// TIA Portal V16 export
// export: Created 2020-03-22T19:23:53.3719267Z, ExportSetting WithDefaults, DisplayName Totally Integrated Automation Portal, DisplayVersion V16, DisplayName TIA Portal Version Control Interface, DisplayVersion V16, DisplayName TIA Portal Openness, DisplayVersion V16, DisplayName TIA Portal Teamcenter Gateway, DisplayVersion V16, DisplayName SINAMICS Startdrive Advanced, DisplayVersion V16 Update 1, DisplayName SINAMICS Startdrive G130, G150, S120, S150, SINAMICS MV, S210, DisplayVersion V16 Update 1, DisplayName SINAMICS Startdrive G110M, G120, G120C, G120D, G120P, DisplayVersion V16 Update 1, DisplayName STEP 7 Professional, DisplayVersion V16, DisplayName STEP 7 Safety, DisplayVersion V16, DisplayName WinCC Professional, DisplayVersion V16
FUNCTION_BLOCK "TX-AI"   // FB804, LAD
{ S7_Optimized_Access := 'TRUE' }
VERSION : 1.0
// stored: AutoNumber false, IsIECCheckEnabled false, IsRetainMemResEnabled false, MemoryReserve 100, SetENOAutomatically false, UDAEnableTagReadback false
   VAR_INPUT
      Mode { ExternalAccessible := 'False'; ExternalVisible := 'False'; ExternalWritable := 'False'} : Int;   // TX Mode - 0 = 4-20 mA / 1 = Int Math (RTD/TC) / 3 = SQRT / 6 = Vortex
      RAIVI { ExternalAccessible := 'False'; ExternalVisible := 'False'; ExternalWritable := 'False'} : Int;   // Raw Analog Input Value INT
      RAIVR { ExternalAccessible := 'False'; ExternalVisible := 'False'; ExternalWritable := 'False'} : Real;   // Raw Analog Input Value REAL
   END_VAR
   VAR_OUTPUT
      SAI : Real;   // Compensated Scaled Analog Value
   END_VAR
   VAR
      HMI : Struct   // Alarms
         Status : Struct
            USAV : Real;   // Uncompensated Scaled Analog Value
            TCV : Real;   // Temperature Compensation Value
            PCV : Real;   // Pressure Compensation Value
            NV : Real;   // Normalized Value
         END_STRUCT;
         Alarm : Struct   // Alarms
            AHHH : Bool;   // Alarm - High High High
            AHH : Bool;   // Alarm - High High
            AH : Bool;   // Alarm - High
            AL : Bool;   // Alarm - Low
            ALL : Bool;   // Alarm - Low Low
            ALLL : Bool;   // Alarm - Low Low Low
            "OR" : Bool;   // Alarm Over Range
            UR : Bool;   // Alarm Under Range
            Fault : Bool;   // Alarm Fault
            SUB : Bool;   // Fault detected and output value is the defined subsitution value
            CH_Fault : Bool;
         END_STRUCT;
         Config : Struct   // Settings
            RIMXV : Real := 27648.0;   // Raw Input Maximum Value (Used for Sqrt)
            RIMNV : Real;   // Raw Input Minimum Value (Used for Sqrt)
            ESMXV : Real := 100.0;   // Engineering/Scaled Maximum Value
            ESMNV : Real;   // Engineering/Scaled Minimum Value
            COV : Bool;   // Clamp Output Value
            OV : Real;   // Offset Value
            SAM : Bool;   // Substitution Activation Mode
            SAV : Real := -999999.0;   // Substitution Value during a limit input value trip
            CE : Struct   // Compensation Equation
               TC : Real := 460.0;   // Temperature Constant
               PC : Real := 14.7;   // Pressure Constant
               TR : Real := 1.0;   // Temperature Reference
               TA : Real := 1.0;   // Temperature Actual
               PR : Real := 1.0;   // Pressure Reference
               PA : Real := 1.0;   // Pressure Actual
            END_STRUCT;
            SP : Struct   // Setpoints
               Limits : Struct
                  HHH : Real := 95.0;   // HHH Limit Setpoint
                  HH : Real := 90.0;   // HH Limit Setpoint
                  H : Real := 80.0;   // HH Limit Setpoint
                  L : Real := 20.0;   // L Limit Setpoint
                  LL : Real := 10.0;   // LL Limit Setpoint
                  LLL : Real := 5.0;   // LLL Limit Setpoint
                  "OR" : Real := 5.0;   // Over range value
                  UR : Real := 5.0;   // Under range value
               END_STRUCT;
               HYS : Struct   // Hysteresis
                  Global : Real;   // Hysteresis global value, only valid when greater than or equal to 0
                  HHH : Real := 1.0;   // Hysteresis Setpoint - High High High
                  HH : Real := 1.0;   // Hysteresis Setpoint - High High
                  H : Real := 1.0;   // Hysteresis Setpoint - High
                  L : Real := 1.0;   // Hysteresis Setpoint - Low
                  LL : Real := 1.0;   // Hysteresis Setpoint - Low Low
                  LLL : Real := 1.0;   // Hysteresis Setpoint - Low Low Low
                  "OR" : Real := 1.0;   // Hysteresis Setpoint - Over Range
                  UR : Real := 1.0;   // Hysteresis Setpoint - Under Range
               END_STRUCT;
               SUB_ON : Bool;   // Substitution Activation
            END_STRUCT;
            PT : Struct   // Setpoints
               HLD : Struct   // Hold
                  Global : Time;   // Hold PT global value, only valid when not equal to 0
                  AHHH : Time := T#1S;   // Alarm Debounce
                  AHH : Time := T#1S;   // Alarm Debounce
                  AH : Time := T#1S;   // Alarm Debounce
                  AL : Time := T#1S;   // Alarm Debounce
                  ALL : Time := T#1S;   // Alarm Debounce
                  ALLL : Time := T#1S;   // Alarm Debounce
                  "OR" : Time := T#1S;   // Over range hold
                  UR : Time := T#1S;   // Under range hold
               END_STRUCT;
               DBNC : Struct   // Debounce
                  Global : Time;   // Debounce PT global value, only valid when not equal to 0
                  AHHH : Time := T#1S;   // Alarm Debounce
                  AHH : Time := T#1S;   // Alarm Debounce
                  AH : Time := T#1S;   // Alarm Debounce
                  AL : Time := T#1S;   // Alarm Debounce
                  ALL : Time := T#1S;   // Alarm Debounce
                  ALLL : Time := T#1S;   // Alarm Debounce
                  "OR" : Time := T#1S;   // Over range debounce
                  UR : Time := T#1S;   // Under range debounce
               END_STRUCT;
            END_STRUCT;
         END_STRUCT;
         Diag : Struct   // Diagnostics
            SV : Real;   // Simulation Value
         END_STRUCT;
      END_STRUCT;
      Admin : Struct   // Admin configurations
         SCL : Struct   // Scale Values
            RDP : Real := 10.0;   // RTD Decimal Places
            RRIMD : Real := 1.0;   // Raw Real input Math divider
            "OR" : Real;   // Over Range Value
            UR : Real;   // Under Range Value
            SAIV : Real;   // Scaled Analog Input Value
         END_STRUCT;
         HYS : Struct   // Hysteresis - Computed Values
            "OR" : Real;   // Hysteresis Value - Over Range
            UR : Real;   // Hysteresis Value - Under Range
         END_STRUCT;
      END_STRUCT;
      OR_DB { ExternalAccessible := 'False'; ExternalVisible := 'False'; ExternalWritable := 'False'} : TON_TIME;   // Over Range Debounce
      UR_DB { ExternalAccessible := 'False'; ExternalVisible := 'False'; ExternalWritable := 'False'} : TON_TIME;   // Under Range DB
      OR_HLD { ExternalAccessible := 'False'; ExternalVisible := 'False'; ExternalWritable := 'False'} : TOF_TIME;   // Over Range Hold
      UR_HLD { ExternalAccessible := 'False'; ExternalVisible := 'False'; ExternalWritable := 'False'} : TOF_TIME;   // Under Range Hold
      HHHA { ExternalAccessible := 'False'; ExternalVisible := 'False'; ExternalWritable := 'False'} : "HLR";   // High High High Alarm
      HHA { ExternalAccessible := 'False'; ExternalVisible := 'False'; ExternalWritable := 'False'} : "HLR";   // High High Alarm
      HA { ExternalAccessible := 'False'; ExternalVisible := 'False'; ExternalWritable := 'False'} : "HLR";   // High Alarm
      LA { ExternalAccessible := 'False'; ExternalVisible := 'False'; ExternalWritable := 'False'} : "LLR";   // Low Alarm
      LLA { ExternalAccessible := 'False'; ExternalVisible := 'False'; ExternalWritable := 'False'} : "LLR";   // Low Low Alarm
      LLLA { ExternalAccessible := 'False'; ExternalVisible := 'False'; ExternalWritable := 'False'} : "LLR";   // Low Low Low Alarm
      molActual { ExternalAccessible := 'False'; ExternalVisible := 'False'; ExternalWritable := 'False'} : Real := 1.0;
      molDesign { ExternalAccessible := 'False'; ExternalVisible := 'False'; ExternalWritable := 'False'} : Real := 1.0;
   END_VAR
   VAR_TEMP
      RAIDI : DInt;   // Raw Analog Input DINT
      RAIR : Real;   // Raw Analog Input REAL
      RAIAV : Real;   // Raw Analog Input Absolute Value
      RAISRV : Real;   // Raw Analog Input Square Root Value
      RAIVS : Real;   // Raw Analog Input Value Scaler
      TCRE : Real;   // Temperature Compensation Reference Equation
      TCAE : Real;   // Temperature Compensation Actual Equation
      PCRE : Real;   // Pressure Compensation Reference Equation
      PCAE : Real;   // Pressure Compensation Actual Equation
      TPCV : Real;   // Temperature Pressure Compensation Value
      MWCV : Real;   // Mol Weight Compensation Value
      TPMCV : Real;   // Temperature Pressure Mol Compensation Value
      sqrtSaiv : Real;   // SCALED ANALOG INT VALUE TO BE SQRT'D
      rawValue : Int;
      dummy : Bool;
      sqrt01 : Real;
      RAIVR_1 : DInt;
      RAIVR_1_1 : Real;
   END_VAR
   VAR_TEMP   // added for the SCL form of the ladder/FBD networks
      _w1 : Bool;
      _w2 : Bool;
   END_VAR
BEGIN

REGION Network 1: Transmitter Mode 1 = Int Math or RTD
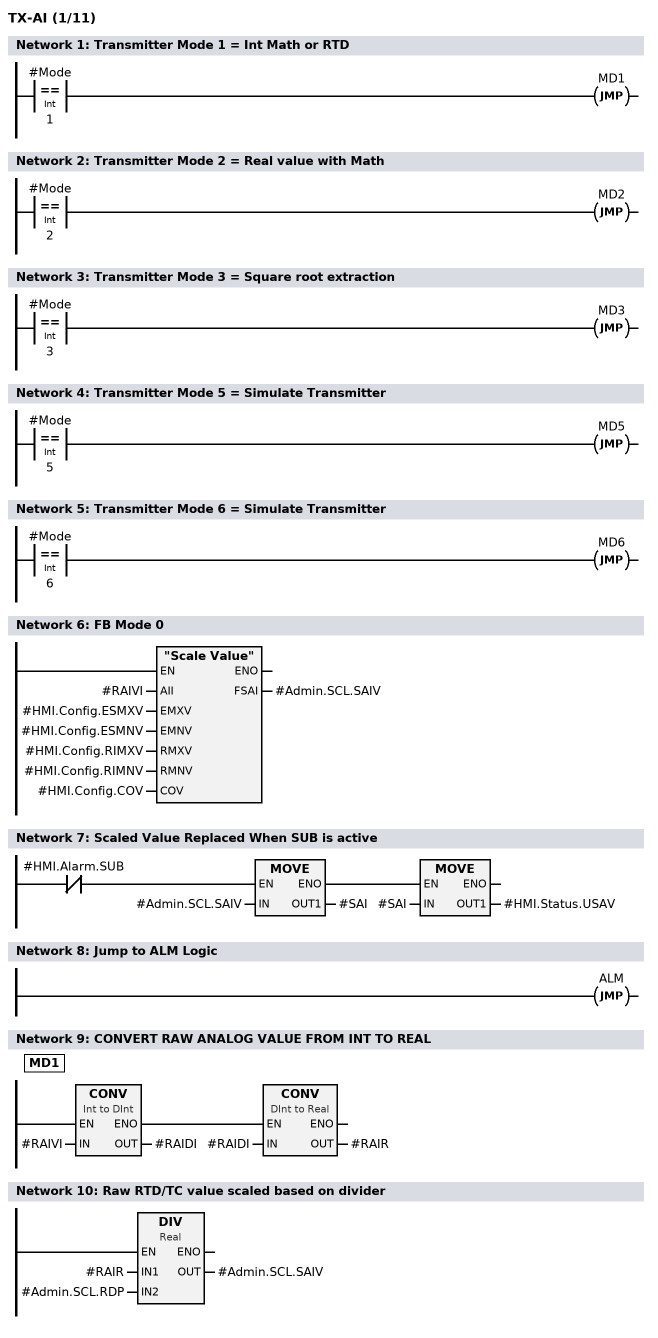
   RUNG wire#powerrail
      { S7_Templates := "SrcType := Int" } EQ_Contact(in1 := #Mode, in2 := 1)
      JumpCoil( MD1 )
   END_RUNG
   // the same network as SCL:
   IF #Mode = 1 THEN GOTO MD1; END_IF;
END_REGION

REGION Network 2: Transmitter Mode 2 = Real value with Math
   RUNG wire#powerrail
      { S7_Templates := "SrcType := Int" } EQ_Contact(in1 := #Mode, in2 := 2)
      JumpCoil( MD2 )
   END_RUNG
   // the same network as SCL:
   IF #Mode = 2 THEN GOTO MD2; END_IF;
END_REGION

REGION Network 3: Transmitter Mode 3 = Square root extraction
   RUNG wire#powerrail
      { S7_Templates := "SrcType := Int" } EQ_Contact(in1 := #Mode, in2 := 3)
      JumpCoil( MD3 )
   END_RUNG
   // the same network as SCL:
   IF #Mode = 3 THEN GOTO MD3; END_IF;
END_REGION

REGION Network 4: Transmitter Mode 5 = Simulate Transmitter
   RUNG wire#powerrail
      { S7_Templates := "SrcType := Int" } EQ_Contact(in1 := #Mode, in2 := 5)
      JumpCoil( MD5 )
   END_RUNG
   // the same network as SCL:
   IF #Mode = 5 THEN GOTO MD5; END_IF;
END_REGION

REGION Network 5: Transmitter Mode 6 = Simulate Transmitter
   RUNG wire#powerrail
      { S7_Templates := "SrcType := Int" } EQ_Contact(in1 := #Mode, in2 := 6)
      JumpCoil( MD6 )
   END_RUNG
   // the same network as SCL:
   IF #Mode = 6 THEN GOTO MD6; END_IF;
END_REGION

REGION Network 6: FB Mode 0
   RUNG wire#powerrail
      "Scale Value"(AII := #RAIVI, EMXV := #HMI.Config.ESMXV, EMNV := #HMI.Config.ESMNV, RMXV := #HMI.Config.RIMXV, RMNV := #HMI.Config.RIMNV, COV := #HMI.Config.COV, FSAI => #Admin.SCL.SAIV)
   END_RUNG
   // the same network as SCL:
   "Scale Value"(AII := #RAIVI,
                 EMXV := #HMI.Config.ESMXV,
                 EMNV := #HMI.Config.ESMNV,
                 RMXV := #HMI.Config.RIMXV,
                 RMNV := #HMI.Config.RIMNV,
                 COV := #HMI.Config.COV,
                 FSAI => #Admin.SCL.SAIV);
END_REGION

REGION Network 7: Scaled Value Replaced When SUB is active
   RUNG wire#powerrail
      I_Contact( #HMI.Alarm.SUB )
      { S7_GenerateENO := "TRUE" } Move(in := #Admin.SCL.SAIV, out1 => #SAI)
      { S7_GenerateENO := "TRUE" } Move(in := #SAI, out1 => #HMI.Status.USAV)
   END_RUNG
   // the same network as SCL:
   // ENO of a box is taken as its EN; it also drops when the box reports an error
   IF NOT #HMI.Alarm.SUB THEN
       #SAI := #Admin.SCL.SAIV;
       #HMI.Status.USAV := #SAI;
   END_IF;
END_REGION

REGION Network 8: Jump to ALM Logic
   RUNG wire#powerrail
      JumpCoil( ALM )
   END_RUNG
   // the same network as SCL:
   GOTO ALM;
END_REGION

REGION Network 9: CONVERT RAW ANALOG VALUE FROM INT TO REAL
   Label( MD1 )
   RUNG wire#powerrail
      { S7_Templates := "[SrcType := Int, DestType := DInt]"; S7_GenerateENO := "TRUE" } Convert(in := #RAIVI, out => #RAIDI)
      { S7_Templates := "[SrcType := DInt, DestType := Real]"; S7_GenerateENO := "TRUE" } Convert(in := #RAIDI, out => #RAIR)
   END_RUNG
   // the same network as SCL:
   // ENO of a box is taken as its EN; it also drops when the box reports an error
   MD1:
   #RAIDI := INT_TO_DINT(#RAIVI);
   #RAIR := DINT_TO_REAL(#RAIDI);
END_REGION

REGION Network 10: Raw RTD/TC value scaled based on divider
   RUNG wire#powerrail
      { S7_Templates := "SrcType := Real"; S7_GenerateENO := "TRUE" } Div(in1 := #RAIR, in2 := #Admin.SCL.RDP, out => #Admin.SCL.SAIV)
   END_RUNG
   // the same network as SCL:
   #Admin.SCL.SAIV := #RAIR / #Admin.SCL.RDP;
END_REGION

REGION Network 11: Scaled Value Replaced When SUB is active
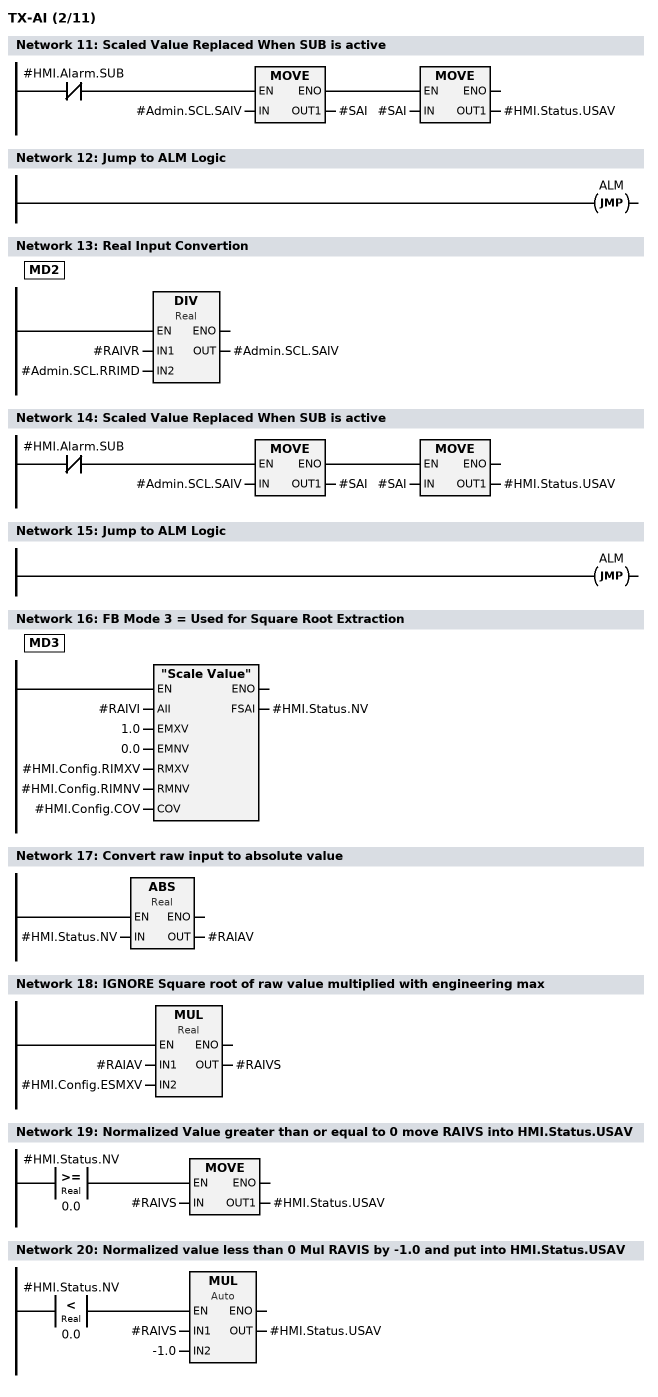
   RUNG wire#powerrail
      I_Contact( #HMI.Alarm.SUB )
      { S7_GenerateENO := "TRUE" } Move(in := #Admin.SCL.SAIV, out1 => #SAI)
      Move(in := #SAI, out1 => #HMI.Status.USAV)
   END_RUNG
   // the same network as SCL:
   // ENO of a box is taken as its EN; it also drops when the box reports an error
   IF NOT #HMI.Alarm.SUB THEN
       #SAI := #Admin.SCL.SAIV;
       #HMI.Status.USAV := #SAI;
   END_IF;
END_REGION

REGION Network 12: Jump to ALM Logic
   RUNG wire#powerrail
      JumpCoil( ALM )
   END_RUNG
   // the same network as SCL:
   GOTO ALM;
END_REGION

REGION Network 13: Real Input Convertion
   Label( MD2 )
   RUNG wire#powerrail
      { S7_Templates := "SrcType := Real"; S7_GenerateENO := "TRUE" } Div(in1 := #RAIVR, in2 := #Admin.SCL.RRIMD, out => #Admin.SCL.SAIV)
   END_RUNG
   // the same network as SCL:
   MD2:
   #Admin.SCL.SAIV := #RAIVR / #Admin.SCL.RRIMD;
END_REGION

REGION Network 14: Scaled Value Replaced When SUB is active
   RUNG wire#powerrail
      I_Contact( #HMI.Alarm.SUB )
      { S7_GenerateENO := "TRUE" } Move(in := #Admin.SCL.SAIV, out1 => #SAI)
      Move(in := #SAI, out1 => #HMI.Status.USAV)
   END_RUNG
   // the same network as SCL:
   // ENO of a box is taken as its EN; it also drops when the box reports an error
   IF NOT #HMI.Alarm.SUB THEN
       #SAI := #Admin.SCL.SAIV;
       #HMI.Status.USAV := #SAI;
   END_IF;
END_REGION

REGION Network 15: Jump to ALM Logic
   RUNG wire#powerrail
      JumpCoil( ALM )
   END_RUNG
   // the same network as SCL:
   GOTO ALM;
END_REGION

REGION Network 16: FB Mode 3 = Used for Square Root Extraction
   Label( MD3 )
   RUNG wire#powerrail
      "Scale Value"(AII := #RAIVI, EMXV := 1.0, EMNV := 0.0, RMXV := #HMI.Config.RIMXV, RMNV := #HMI.Config.RIMNV, COV := #HMI.Config.COV, FSAI => #HMI.Status.NV)
   END_RUNG
   // the same network as SCL:
   MD3:
   "Scale Value"(AII := #RAIVI,
                 EMXV := 1.0,
                 EMNV := 0.0,
                 RMXV := #HMI.Config.RIMXV,
                 RMNV := #HMI.Config.RIMNV,
                 COV := #HMI.Config.COV,
                 FSAI => #HMI.Status.NV);
END_REGION

REGION Network 17: Convert raw input to absolute value
   RUNG wire#powerrail
      { S7_Templates := "SrcType := Real"; S7_GenerateENO := "TRUE" } Abs(in := #HMI.Status.NV, out => #RAIAV)
   END_RUNG
   // the same network as SCL:
   #RAIAV := ABS(#HMI.Status.NV);
END_REGION

REGION Network 18: IGNORE Square root of raw value multiplied with engineering max
   RUNG wire#powerrail
      { S7_Templates := "SrcType := Real"; S7_GenerateENO := "TRUE" } Mul(in1 := #RAIAV, in2 := #HMI.Config.ESMXV, out => #RAIVS)
   END_RUNG
   // the same network as SCL:
   #RAIVS := #RAIAV * #HMI.Config.ESMXV;
END_REGION

REGION Network 19: Normalized Value greater than or equal to 0 move RAIVS into HMI.Status.USAV
   RUNG wire#powerrail
      { S7_Templates := "SrcType := Real" } GE_Contact(in1 := #HMI.Status.NV, in2 := 0.0)
      { S7_GenerateENO := "TRUE" } Move(in := #RAIVS, out1 => #HMI.Status.USAV)
   END_RUNG
   // the same network as SCL:
   IF #HMI.Status.NV >= 0.0 THEN #HMI.Status.USAV := #RAIVS; END_IF;
END_REGION

REGION Network 20: Normalized value less than 0 Mul RAVIS by -1.0 and put into HMI.Status.USAV
   RUNG wire#powerrail
      { S7_Templates := "SrcType := Real" } LT_Contact(in1 := #HMI.Status.NV, in2 := 0.0)
      { S7_GenerateENO := "TRUE" } Mul(in1 := #RAIVS, in2 := -1.0, out => #HMI.Status.USAV)
   END_RUNG
   // the same network as SCL:
   IF #HMI.Status.NV < 0.0 THEN #HMI.Status.USAV := #RAIVS * (-1.0); END_IF;
END_REGION

REGION Network 21: Temperature Compensation Equation Step 1
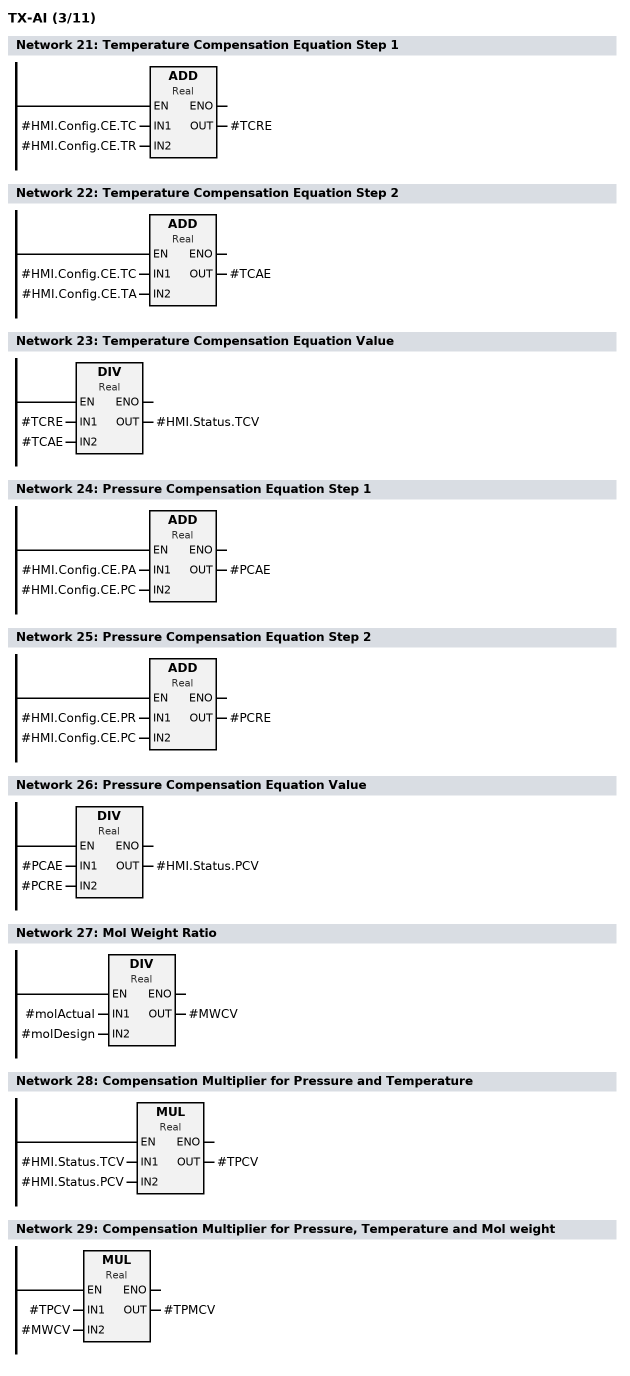
   RUNG wire#powerrail
      { S7_Templates := "SrcType := Real"; S7_GenerateENO := "TRUE" } Add(in1 := #HMI.Config.CE.TC, in2 := #HMI.Config.CE.TR, out => #TCRE)
   END_RUNG
   // the same network as SCL:
   #TCRE := #HMI.Config.CE.TC + #HMI.Config.CE.TR;
END_REGION

REGION Network 22: Temperature Compensation Equation Step 2
   RUNG wire#powerrail
      { S7_Templates := "SrcType := Real"; S7_GenerateENO := "TRUE" } Add(in1 := #HMI.Config.CE.TC, in2 := #HMI.Config.CE.TA, out => #TCAE)
   END_RUNG
   // the same network as SCL:
   #TCAE := #HMI.Config.CE.TC + #HMI.Config.CE.TA;
END_REGION

REGION Network 23: Temperature Compensation Equation Value
   RUNG wire#powerrail
      { S7_Templates := "SrcType := Real"; S7_GenerateENO := "TRUE" } Div(in1 := #TCRE, in2 := #TCAE, out => #HMI.Status.TCV)
   END_RUNG
   // the same network as SCL:
   #HMI.Status.TCV := #TCRE / #TCAE;
END_REGION

REGION Network 24: Pressure Compensation Equation Step 1
   RUNG wire#powerrail
      { S7_Templates := "SrcType := Real"; S7_GenerateENO := "TRUE" } Add(in1 := #HMI.Config.CE.PA, in2 := #HMI.Config.CE.PC, out => #PCAE)
   END_RUNG
   // the same network as SCL:
   #PCAE := #HMI.Config.CE.PA + #HMI.Config.CE.PC;
END_REGION

REGION Network 25: Pressure Compensation Equation Step 2
   RUNG wire#powerrail
      { S7_Templates := "SrcType := Real"; S7_GenerateENO := "TRUE" } Add(in1 := #HMI.Config.CE.PR, in2 := #HMI.Config.CE.PC, out => #PCRE)
   END_RUNG
   // the same network as SCL:
   #PCRE := #HMI.Config.CE.PR + #HMI.Config.CE.PC;
END_REGION

REGION Network 26: Pressure Compensation Equation Value
   RUNG wire#powerrail
      { S7_Templates := "SrcType := Real"; S7_GenerateENO := "TRUE" } Div(in1 := #PCAE, in2 := #PCRE, out => #HMI.Status.PCV)
   END_RUNG
   // the same network as SCL:
   #HMI.Status.PCV := #PCAE / #PCRE;
END_REGION

REGION Network 27: Mol Weight Ratio
   RUNG wire#powerrail
      { S7_Templates := "SrcType := Real"; S7_GenerateENO := "TRUE" } Div(in1 := #molActual, in2 := #molDesign, out => #MWCV)
   END_RUNG
   // the same network as SCL:
   #MWCV := #molActual / #molDesign;
END_REGION

REGION Network 28: Compensation Multiplier for Pressure and Temperature
   RUNG wire#powerrail
      { S7_Templates := "SrcType := Real"; S7_GenerateENO := "TRUE" } Mul(in1 := #HMI.Status.TCV, in2 := #HMI.Status.PCV, out => #TPCV)
   END_RUNG
   // the same network as SCL:
   #TPCV := #HMI.Status.TCV * #HMI.Status.PCV;
END_REGION

REGION Network 29: Compensation Multiplier for Pressure, Temperature and Mol weight
   RUNG wire#powerrail
      { S7_Templates := "SrcType := Real"; S7_GenerateENO := "TRUE" } Mul(in1 := #TPCV, in2 := #MWCV, out => #TPMCV)
   END_RUNG
   // the same network as SCL:
   #TPMCV := #TPCV * #MWCV;
END_REGION

REGION Network 30: Compensated Analog Value
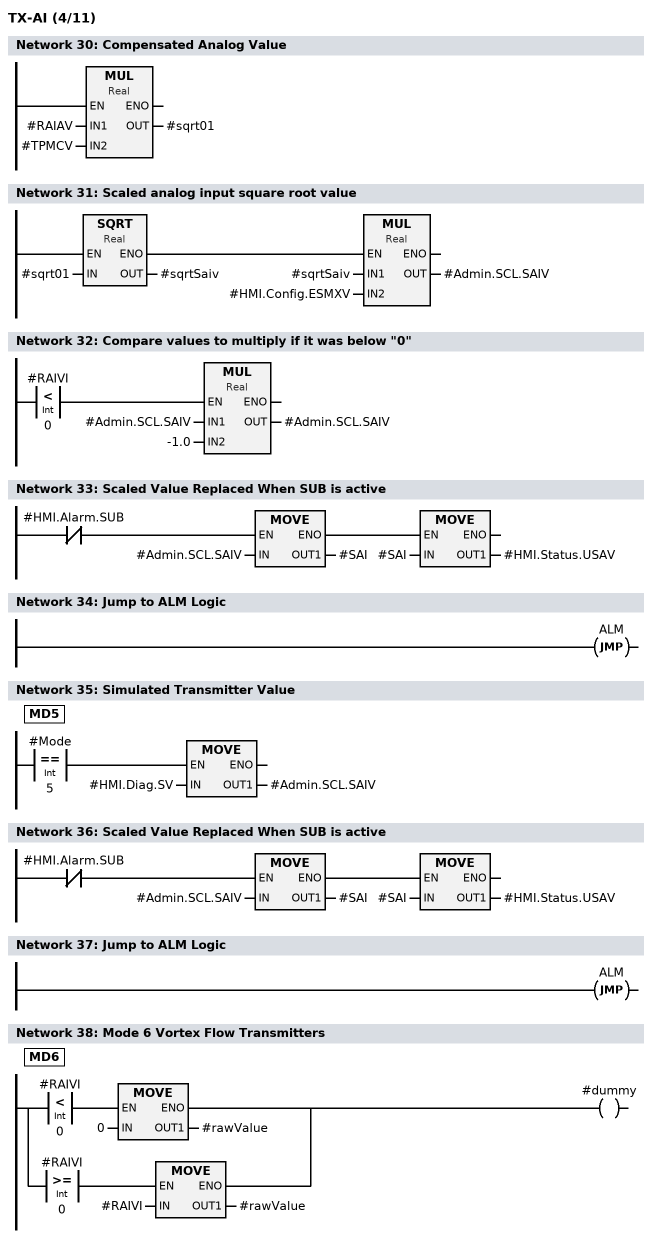
   RUNG wire#powerrail
      { S7_Templates := "SrcType := Real"; S7_GenerateENO := "TRUE" } Mul(in1 := #RAIAV, in2 := #TPMCV, out => #sqrt01)
   END_RUNG
   // the same network as SCL:
   #sqrt01 := #RAIAV * #TPMCV;
END_REGION

REGION Network 31: Scaled analog input square root value
   // ENO of a box is taken as its EN; it also drops when the box reports an error
   #sqrtSaiv := SQRT(#sqrt01);
   #Admin.SCL.SAIV := #sqrtSaiv * #HMI.Config.ESMXV;
END_REGION

REGION Network 32: Compare values to multiply if it was below "0"
   RUNG wire#powerrail
      { S7_Templates := "SrcType := Int" } LT_Contact(in1 := #RAIVI, in2 := 0)
      { S7_Templates := "SrcType := Real"; S7_GenerateENO := "TRUE" } Mul(in1 := #Admin.SCL.SAIV, in2 := -1.0, out => #Admin.SCL.SAIV)
   END_RUNG
   // the same network as SCL:
   IF #RAIVI < 0 THEN #Admin.SCL.SAIV := #Admin.SCL.SAIV * (-1.0); END_IF;
END_REGION

REGION Network 33: Scaled Value Replaced When SUB is active
   RUNG wire#powerrail
      I_Contact( #HMI.Alarm.SUB )
      { S7_GenerateENO := "TRUE" } Move(in := #Admin.SCL.SAIV, out1 => #SAI)
      { S7_GenerateENO := "TRUE" } Move(in := #SAI, out1 => #HMI.Status.USAV)
   END_RUNG
   // the same network as SCL:
   // ENO of a box is taken as its EN; it also drops when the box reports an error
   IF NOT #HMI.Alarm.SUB THEN
       #SAI := #Admin.SCL.SAIV;
       #HMI.Status.USAV := #SAI;
   END_IF;
END_REGION

REGION Network 34: Jump to ALM Logic
   RUNG wire#powerrail
      JumpCoil( ALM )
   END_RUNG
   // the same network as SCL:
   GOTO ALM;
END_REGION

REGION Network 35: Simulated Transmitter Value
   Label( MD5 )
   RUNG wire#powerrail
      { S7_Templates := "SrcType := Int" } EQ_Contact(in1 := #Mode, in2 := 5)
      { S7_GenerateENO := "TRUE" } Move(in := #HMI.Diag.SV, out1 => #Admin.SCL.SAIV)
   END_RUNG
   // the same network as SCL:
   MD5:
   IF #Mode = 5 THEN #Admin.SCL.SAIV := #HMI.Diag.SV; END_IF;
END_REGION

REGION Network 36: Scaled Value Replaced When SUB is active
   RUNG wire#powerrail
      I_Contact( #HMI.Alarm.SUB )
      { S7_GenerateENO := "TRUE" } Move(in := #Admin.SCL.SAIV, out1 => #SAI)
      { S7_GenerateENO := "TRUE" } Move(in := #SAI, out1 => #HMI.Status.USAV)
   END_RUNG
   // the same network as SCL:
   // ENO of a box is taken as its EN; it also drops when the box reports an error
   IF NOT #HMI.Alarm.SUB THEN
       #SAI := #Admin.SCL.SAIV;
       #HMI.Status.USAV := #SAI;
   END_IF;
END_REGION

REGION Network 37: Jump to ALM Logic
   RUNG wire#powerrail
      JumpCoil( ALM )
   END_RUNG
   // the same network as SCL:
   GOTO ALM;
END_REGION

REGION Network 38: Mode 6 Vortex Flow Transmitters
   Label( MD6 )
   RUNG wire#powerrail
      { S7_Templates := "SrcType := Int" } LT_Contact(in1 := #RAIVI, in2 := 0)
      { S7_GenerateENO := "TRUE" } Move(in := 0, out1 => #rawValue)
      wire#w1
      Coil( #dummy )
   END_RUNG
   RUNG wire#powerrail
      { S7_Templates := "SrcType := Int" } GE_Contact(in1 := #RAIVI, in2 := 0)
      { S7_GenerateENO := "TRUE" } Move(in := #RAIVI, out1 => #rawValue)
   END_RUNG wire#w1
   // the same network as SCL:
   // ENO of a box is taken as its EN; it also drops when the box reports an error
   MD6:
   #_w1 := #RAIVI < 0;
   IF #_w1 THEN #rawValue := 0; END_IF;
   #_w2 := #RAIVI >= 0;
   IF #_w2 THEN #rawValue := #RAIVI; END_IF;
   #dummy := #_w1 OR #_w2;
END_REGION

REGION Network 39: Normalize signal 4-20mA to 0-1 ratio
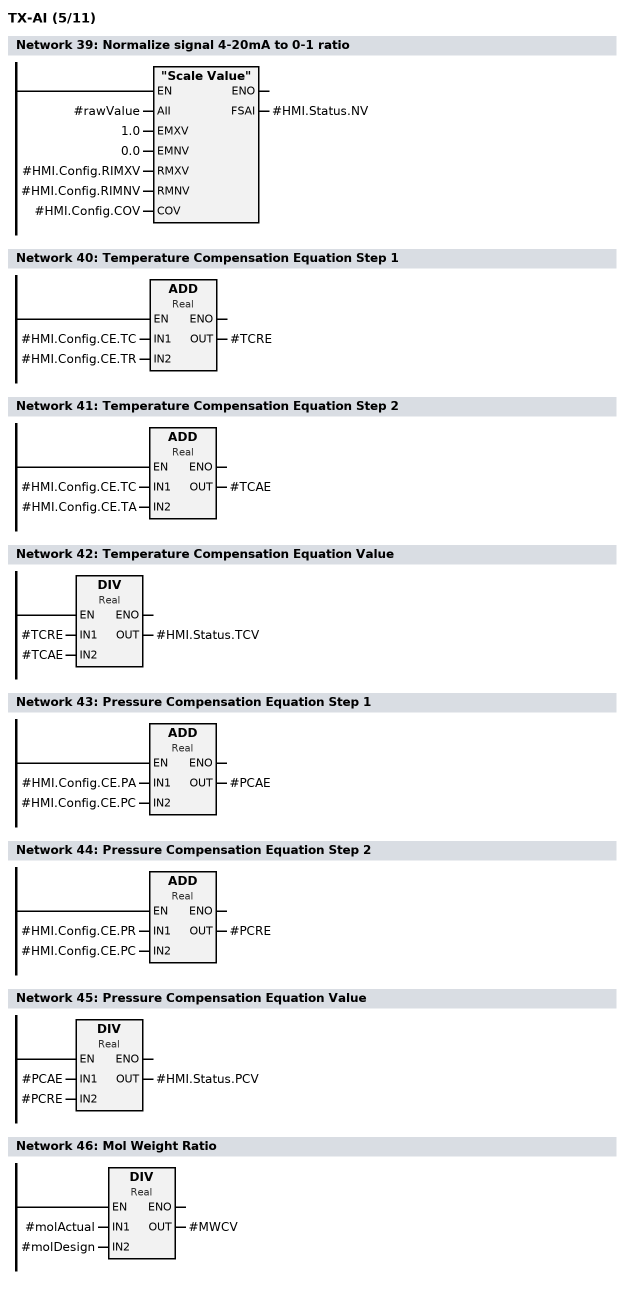
   RUNG wire#powerrail
      "Scale Value"(AII := #rawValue, EMXV := 1.0, EMNV := 0.0, RMXV := #HMI.Config.RIMXV, RMNV := #HMI.Config.RIMNV, COV := #HMI.Config.COV, FSAI => #HMI.Status.NV)
   END_RUNG
   // the same network as SCL:
   "Scale Value"(AII := #rawValue,
                 EMXV := 1.0,
                 EMNV := 0.0,
                 RMXV := #HMI.Config.RIMXV,
                 RMNV := #HMI.Config.RIMNV,
                 COV := #HMI.Config.COV,
                 FSAI => #HMI.Status.NV);
END_REGION

REGION Network 40: Temperature Compensation Equation Step 1
   RUNG wire#powerrail
      { S7_Templates := "SrcType := Real"; S7_GenerateENO := "TRUE" } Add(in1 := #HMI.Config.CE.TC, in2 := #HMI.Config.CE.TR, out => #TCRE)
   END_RUNG
   // the same network as SCL:
   #TCRE := #HMI.Config.CE.TC + #HMI.Config.CE.TR;
END_REGION

REGION Network 41: Temperature Compensation Equation Step 2
   RUNG wire#powerrail
      { S7_Templates := "SrcType := Real"; S7_GenerateENO := "TRUE" } Add(in1 := #HMI.Config.CE.TC, in2 := #HMI.Config.CE.TA, out => #TCAE)
   END_RUNG
   // the same network as SCL:
   #TCAE := #HMI.Config.CE.TC + #HMI.Config.CE.TA;
END_REGION

REGION Network 42: Temperature Compensation Equation Value
   RUNG wire#powerrail
      { S7_Templates := "SrcType := Real"; S7_GenerateENO := "TRUE" } Div(in1 := #TCRE, in2 := #TCAE, out => #HMI.Status.TCV)
   END_RUNG
   // the same network as SCL:
   #HMI.Status.TCV := #TCRE / #TCAE;
END_REGION

REGION Network 43: Pressure Compensation Equation Step 1
   RUNG wire#powerrail
      { S7_Templates := "SrcType := Real"; S7_GenerateENO := "TRUE" } Add(in1 := #HMI.Config.CE.PA, in2 := #HMI.Config.CE.PC, out => #PCAE)
   END_RUNG
   // the same network as SCL:
   #PCAE := #HMI.Config.CE.PA + #HMI.Config.CE.PC;
END_REGION

REGION Network 44: Pressure Compensation Equation Step 2
   RUNG wire#powerrail
      { S7_Templates := "SrcType := Real"; S7_GenerateENO := "TRUE" } Add(in1 := #HMI.Config.CE.PR, in2 := #HMI.Config.CE.PC, out => #PCRE)
   END_RUNG
   // the same network as SCL:
   #PCRE := #HMI.Config.CE.PR + #HMI.Config.CE.PC;
END_REGION

REGION Network 45: Pressure Compensation Equation Value
   RUNG wire#powerrail
      { S7_Templates := "SrcType := Real"; S7_GenerateENO := "TRUE" } Div(in1 := #PCAE, in2 := #PCRE, out => #HMI.Status.PCV)
   END_RUNG
   // the same network as SCL:
   #HMI.Status.PCV := #PCAE / #PCRE;
END_REGION

REGION Network 46: Mol Weight Ratio
   RUNG wire#powerrail
      { S7_Templates := "SrcType := Real"; S7_GenerateENO := "TRUE" } Div(in1 := #molActual, in2 := #molDesign, out => #MWCV)
   END_RUNG
   // the same network as SCL:
   #MWCV := #molActual / #molDesign;
END_REGION

REGION Network 47: Compensation Multiplier for Pressure and Temperature
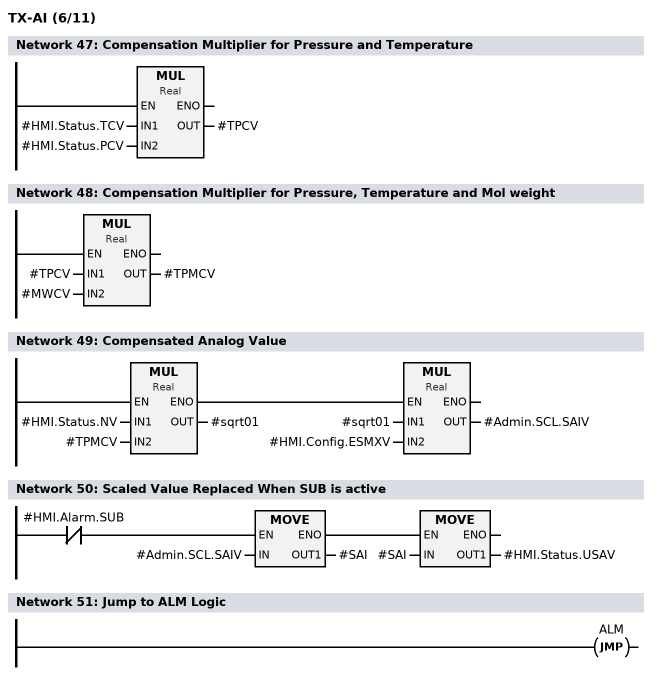
   RUNG wire#powerrail
      { S7_Templates := "SrcType := Real"; S7_GenerateENO := "TRUE" } Mul(in1 := #HMI.Status.TCV, in2 := #HMI.Status.PCV, out => #TPCV)
   END_RUNG
   // the same network as SCL:
   #TPCV := #HMI.Status.TCV * #HMI.Status.PCV;
END_REGION

REGION Network 48: Compensation Multiplier for Pressure, Temperature and Mol weight
   RUNG wire#powerrail
      { S7_Templates := "SrcType := Real"; S7_GenerateENO := "TRUE" } Mul(in1 := #TPCV, in2 := #MWCV, out => #TPMCV)
   END_RUNG
   // the same network as SCL:
   #TPMCV := #TPCV * #MWCV;
END_REGION

REGION Network 49: Compensated Analog Value
   RUNG wire#powerrail
      { S7_Templates := "SrcType := Real"; S7_GenerateENO := "TRUE" } Mul(in1 := #HMI.Status.NV, in2 := #TPMCV, out => #sqrt01)
      { S7_Templates := "SrcType := Real"; S7_GenerateENO := "TRUE" } Mul(in1 := #sqrt01, in2 := #HMI.Config.ESMXV, out => #Admin.SCL.SAIV)
   END_RUNG
   // the same network as SCL:
   // ENO of a box is taken as its EN; it also drops when the box reports an error
   #sqrt01 := #HMI.Status.NV * #TPMCV;
   #Admin.SCL.SAIV := #sqrt01 * #HMI.Config.ESMXV;
END_REGION

REGION Network 50: Scaled Value Replaced When SUB is active
   RUNG wire#powerrail
      I_Contact( #HMI.Alarm.SUB )
      { S7_GenerateENO := "TRUE" } Move(in := #Admin.SCL.SAIV, out1 => #SAI)
      { S7_GenerateENO := "TRUE" } Move(in := #SAI, out1 => #HMI.Status.USAV)
   END_RUNG
   // the same network as SCL:
   // ENO of a box is taken as its EN; it also drops when the box reports an error
   IF NOT #HMI.Alarm.SUB THEN
       #SAI := #Admin.SCL.SAIV;
       #HMI.Status.USAV := #SAI;
   END_IF;
END_REGION

REGION Network 51: Jump to ALM Logic
   RUNG wire#powerrail
      JumpCoil( ALM )
   END_RUNG
   // the same network as SCL:
   GOTO ALM;
END_REGION

REGION Network 52: Global Hold Preset Time Condition
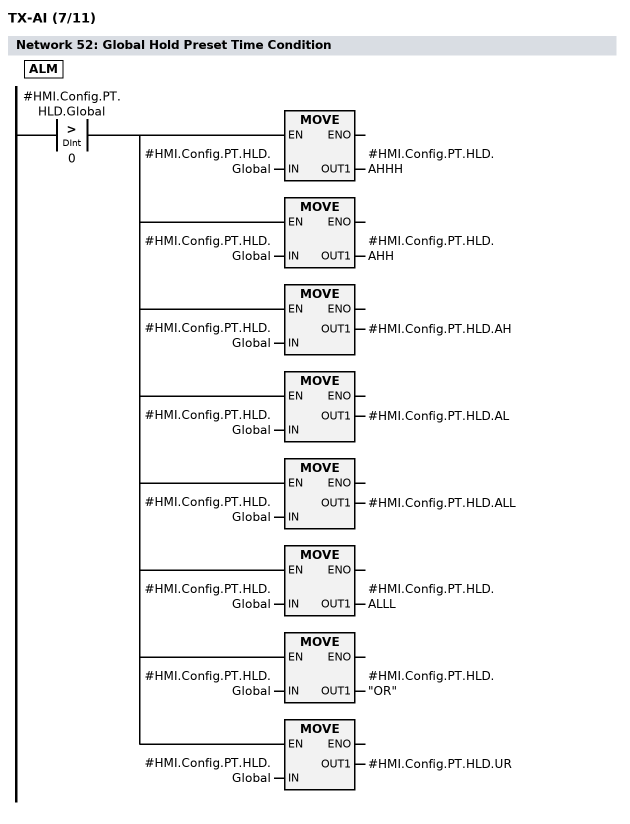
   Label( ALM )
   RUNG wire#powerrail
      { S7_Templates := "SrcType := DInt" } GT_Contact(in1 := #HMI.Config.PT.HLD.Global, in2 := 0)
      wire#w1
      { S7_GenerateENO := "TRUE" } Move(in := #HMI.Config.PT.HLD.Global, out1 => #HMI.Config.PT.HLD.AHHH)
   END_RUNG
   RUNG wire#w1
      { S7_GenerateENO := "TRUE" } Move(in := #HMI.Config.PT.HLD.Global, out1 => #HMI.Config.PT.HLD.AHH)
   END_RUNG
   RUNG wire#w1
      { S7_GenerateENO := "TRUE" } Move(in := #HMI.Config.PT.HLD.Global, out1 => #HMI.Config.PT.HLD.AH)
   END_RUNG
   RUNG wire#w1
      { S7_GenerateENO := "TRUE" } Move(in := #HMI.Config.PT.HLD.Global, out1 => #HMI.Config.PT.HLD.AL)
   END_RUNG
   RUNG wire#w1
      { S7_GenerateENO := "TRUE" } Move(in := #HMI.Config.PT.HLD.Global, out1 => #HMI.Config.PT.HLD.ALL)
   END_RUNG
   RUNG wire#w1
      { S7_GenerateENO := "TRUE" } Move(in := #HMI.Config.PT.HLD.Global, out1 => #HMI.Config.PT.HLD.ALLL)
   END_RUNG
   RUNG wire#w1
      { S7_GenerateENO := "TRUE" } Move(in := #HMI.Config.PT.HLD.Global, out1 => #HMI.Config.PT.HLD."OR")
   END_RUNG
   RUNG wire#w1
      { S7_GenerateENO := "TRUE" } Move(in := #HMI.Config.PT.HLD.Global, out1 => #HMI.Config.PT.HLD.UR)
   END_RUNG
   // the same network as SCL:
   ALM:
   IF #HMI.Config.PT.HLD.Global > 0 THEN
       #HMI.Config.PT.HLD.AHHH := #HMI.Config.PT.HLD.Global;
       #HMI.Config.PT.HLD.AHH := #HMI.Config.PT.HLD.Global;
       #HMI.Config.PT.HLD.AH := #HMI.Config.PT.HLD.Global;
       #HMI.Config.PT.HLD.AL := #HMI.Config.PT.HLD.Global;
       #HMI.Config.PT.HLD.ALL := #HMI.Config.PT.HLD.Global;
       #HMI.Config.PT.HLD.ALLL := #HMI.Config.PT.HLD.Global;
       #HMI.Config.PT.HLD."OR" := #HMI.Config.PT.HLD.Global;
       #HMI.Config.PT.HLD.UR := #HMI.Config.PT.HLD.Global;
   END_IF;
END_REGION

REGION Network 53: Global Debounce Preset Time Condition
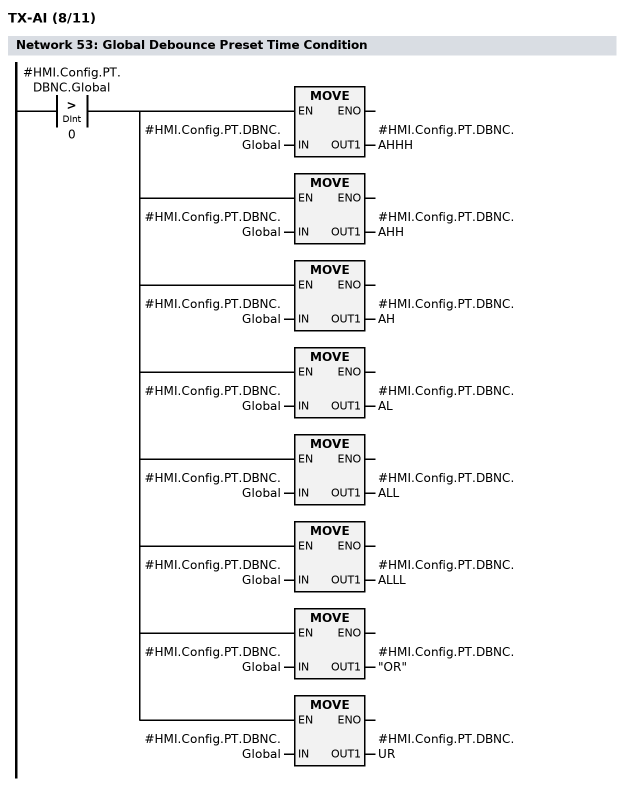
   RUNG wire#powerrail
      { S7_Templates := "SrcType := DInt" } GT_Contact(in1 := #HMI.Config.PT.DBNC.Global, in2 := 0)
      wire#w1
      { S7_GenerateENO := "TRUE" } Move(in := #HMI.Config.PT.DBNC.Global, out1 => #HMI.Config.PT.DBNC.AHHH)
   END_RUNG
   RUNG wire#w1
      { S7_GenerateENO := "TRUE" } Move(in := #HMI.Config.PT.DBNC.Global, out1 => #HMI.Config.PT.DBNC.AHH)
   END_RUNG
   RUNG wire#w1
      { S7_GenerateENO := "TRUE" } Move(in := #HMI.Config.PT.DBNC.Global, out1 => #HMI.Config.PT.DBNC.AH)
   END_RUNG
   RUNG wire#w1
      { S7_GenerateENO := "TRUE" } Move(in := #HMI.Config.PT.DBNC.Global, out1 => #HMI.Config.PT.DBNC.AL)
   END_RUNG
   RUNG wire#w1
      { S7_GenerateENO := "TRUE" } Move(in := #HMI.Config.PT.DBNC.Global, out1 => #HMI.Config.PT.DBNC.ALL)
   END_RUNG
   RUNG wire#w1
      { S7_GenerateENO := "TRUE" } Move(in := #HMI.Config.PT.DBNC.Global, out1 => #HMI.Config.PT.DBNC.ALLL)
   END_RUNG
   RUNG wire#w1
      { S7_GenerateENO := "TRUE" } Move(in := #HMI.Config.PT.DBNC.Global, out1 => #HMI.Config.PT.DBNC."OR")
   END_RUNG
   RUNG wire#w1
      { S7_GenerateENO := "TRUE" } Move(in := #HMI.Config.PT.DBNC.Global, out1 => #HMI.Config.PT.DBNC.UR)
   END_RUNG
   // the same network as SCL:
   IF #HMI.Config.PT.DBNC.Global > 0 THEN
       #HMI.Config.PT.DBNC.AHHH := #HMI.Config.PT.DBNC.Global;
       #HMI.Config.PT.DBNC.AHH := #HMI.Config.PT.DBNC.Global;
       #HMI.Config.PT.DBNC.AH := #HMI.Config.PT.DBNC.Global;
       #HMI.Config.PT.DBNC.AL := #HMI.Config.PT.DBNC.Global;
       #HMI.Config.PT.DBNC.ALL := #HMI.Config.PT.DBNC.Global;
       #HMI.Config.PT.DBNC.ALLL := #HMI.Config.PT.DBNC.Global;
       #HMI.Config.PT.DBNC."OR" := #HMI.Config.PT.DBNC.Global;
       #HMI.Config.PT.DBNC.UR := #HMI.Config.PT.DBNC.Global;
   END_IF;
END_REGION

REGION Network 54: Global Hysteresis Setpoint Condition
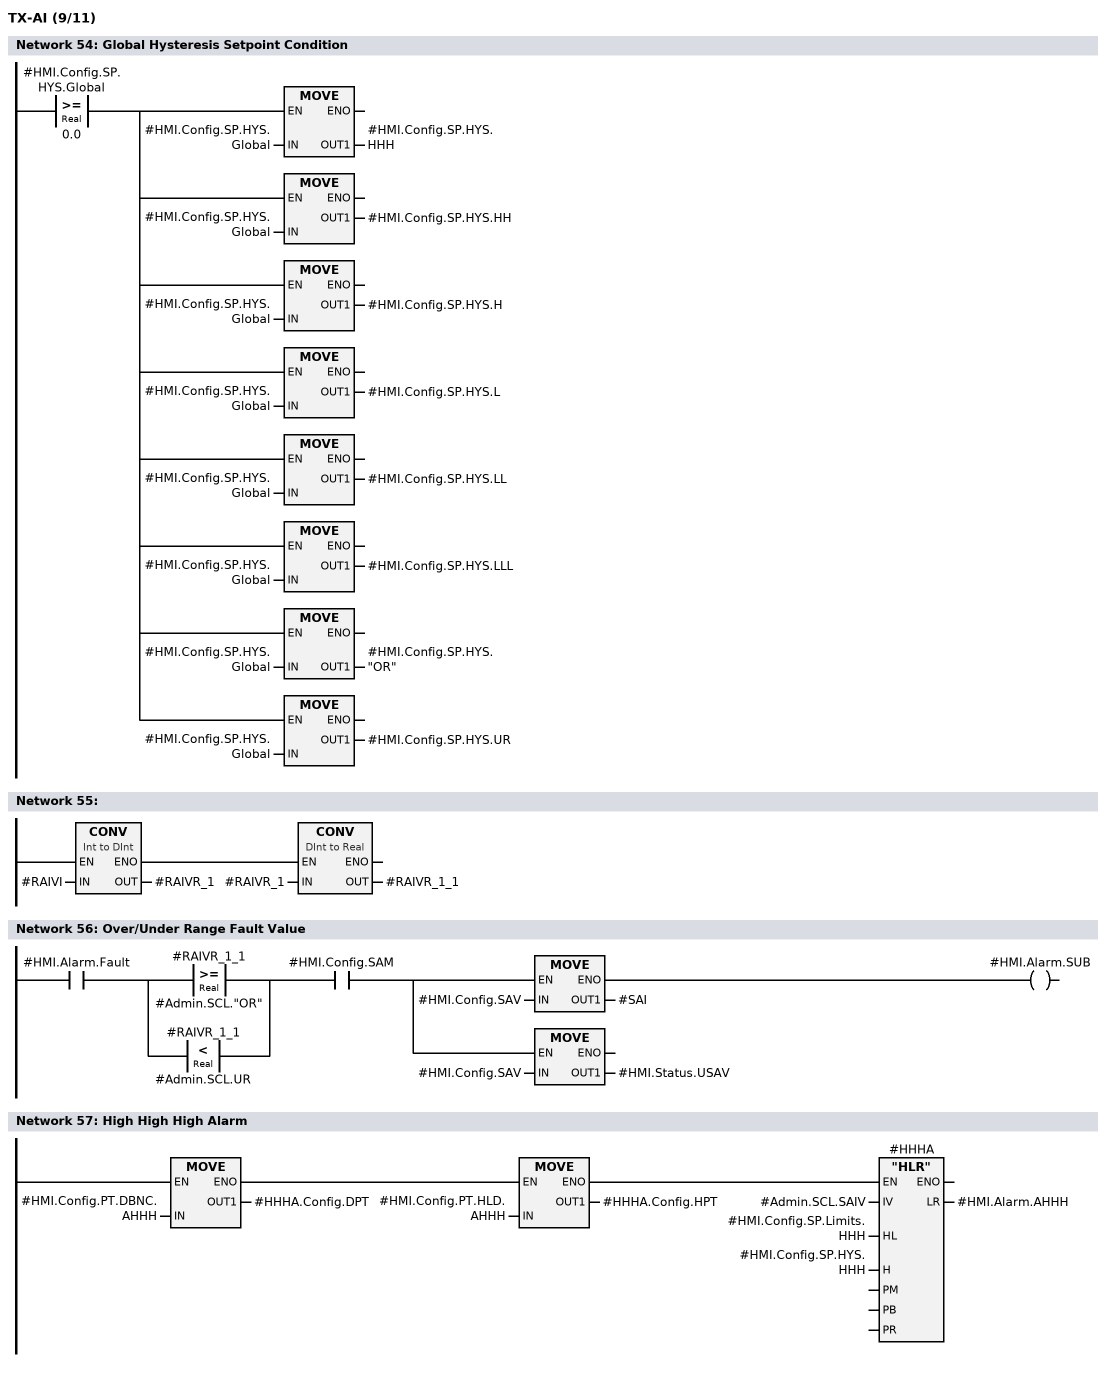
   RUNG wire#powerrail
      { S7_Templates := "SrcType := Real" } GE_Contact(in1 := #HMI.Config.SP.HYS.Global, in2 := 0.0)
      wire#w1
      { S7_GenerateENO := "TRUE" } Move(in := #HMI.Config.SP.HYS.Global, out1 => #HMI.Config.SP.HYS.HHH)
   END_RUNG
   RUNG wire#w1
      { S7_GenerateENO := "TRUE" } Move(in := #HMI.Config.SP.HYS.Global, out1 => #HMI.Config.SP.HYS.HH)
   END_RUNG
   RUNG wire#w1
      { S7_GenerateENO := "TRUE" } Move(in := #HMI.Config.SP.HYS.Global, out1 => #HMI.Config.SP.HYS.H)
   END_RUNG
   RUNG wire#w1
      { S7_GenerateENO := "TRUE" } Move(in := #HMI.Config.SP.HYS.Global, out1 => #HMI.Config.SP.HYS.L)
   END_RUNG
   RUNG wire#w1
      { S7_GenerateENO := "TRUE" } Move(in := #HMI.Config.SP.HYS.Global, out1 => #HMI.Config.SP.HYS.LL)
   END_RUNG
   RUNG wire#w1
      { S7_GenerateENO := "TRUE" } Move(in := #HMI.Config.SP.HYS.Global, out1 => #HMI.Config.SP.HYS.LLL)
   END_RUNG
   RUNG wire#w1
      { S7_GenerateENO := "TRUE" } Move(in := #HMI.Config.SP.HYS.Global, out1 => #HMI.Config.SP.HYS."OR")
   END_RUNG
   RUNG wire#w1
      { S7_GenerateENO := "TRUE" } Move(in := #HMI.Config.SP.HYS.Global, out1 => #HMI.Config.SP.HYS.UR)
   END_RUNG
   // the same network as SCL:
   IF #HMI.Config.SP.HYS.Global >= 0.0 THEN
       #HMI.Config.SP.HYS.HHH := #HMI.Config.SP.HYS.Global;
       #HMI.Config.SP.HYS.HH := #HMI.Config.SP.HYS.Global;
       #HMI.Config.SP.HYS.H := #HMI.Config.SP.HYS.Global;
       #HMI.Config.SP.HYS.L := #HMI.Config.SP.HYS.Global;
       #HMI.Config.SP.HYS.LL := #HMI.Config.SP.HYS.Global;
       #HMI.Config.SP.HYS.LLL := #HMI.Config.SP.HYS.Global;
       #HMI.Config.SP.HYS."OR" := #HMI.Config.SP.HYS.Global;
       #HMI.Config.SP.HYS.UR := #HMI.Config.SP.HYS.Global;
   END_IF;
END_REGION

REGION Network 55
   RUNG wire#powerrail
      { S7_Templates := "[SrcType := Int, DestType := DInt]"; S7_GenerateENO := "TRUE" } Convert(in := #RAIVI, out => #RAIVR_1)
      { S7_Templates := "[SrcType := DInt, DestType := Real]"; S7_GenerateENO := "TRUE" } Convert(in := #RAIVR_1, out => #RAIVR_1_1)
   END_RUNG
   // the same network as SCL:
   // ENO of a box is taken as its EN; it also drops when the box reports an error
   #RAIVR_1 := INT_TO_DINT(#RAIVI);
   #RAIVR_1_1 := DINT_TO_REAL(#RAIVR_1);
END_REGION

REGION Network 56: Over/Under Range Fault Value
   RUNG wire#powerrail
      Contact( #HMI.Alarm.Fault )
      wire#w1
      { S7_Templates := "SrcType := Real" } GE_Contact(in1 := #RAIVR_1_1, in2 := #Admin.SCL."OR")
      wire#w2
      Contact( #HMI.Config.SAM )
      wire#w3
      { S7_GenerateENO := "TRUE" } Move(in := #HMI.Config.SAV, out1 => #SAI)
      Coil( #HMI.Alarm.SUB )
   END_RUNG
   RUNG wire#w1
      { S7_Templates := "SrcType := Real" } LT_Contact(in1 := #RAIVR_1_1, in2 := #Admin.SCL.UR)
   END_RUNG wire#w2
   RUNG wire#w3
      { S7_GenerateENO := "TRUE" } Move(in := #HMI.Config.SAV, out1 => #HMI.Status.USAV)
   END_RUNG
   // the same network as SCL:
   // ENO of a box is taken as its EN; it also drops when the box reports an error
   #_w1 := #HMI.Alarm.Fault AND ((#RAIVR_1_1 >= #Admin.SCL."OR") OR (#RAIVR_1_1 < #Admin.SCL.UR)) AND #HMI.Config.SAM;
   IF #_w1 THEN #SAI := #HMI.Config.SAV; END_IF;
   #HMI.Alarm.SUB := #_w1;
   IF #_w1 THEN #HMI.Status.USAV := #HMI.Config.SAV; END_IF;
END_REGION

REGION Network 57: High High High Alarm
   RUNG wire#powerrail
      { S7_GenerateENO := "TRUE" } Move(in := #HMI.Config.PT.DBNC.AHHH, out1 => #HHHA.Config.DPT)
      { S7_GenerateENO := "TRUE" } Move(in := #HMI.Config.PT.HLD.AHHH, out1 => #HHHA.Config.HPT)
      #HHHA(IV := #Admin.SCL.SAIV, HL := #HMI.Config.SP.Limits.HHH, H := #HMI.Config.SP.HYS.HHH, PM :=, PB :=, PR :=, LR => #HMI.Alarm.AHHH)
   END_RUNG
   // the same network as SCL:
   // ENO of a box is taken as its EN; it also drops when the box reports an error
   #HHHA.Config.DPT := #HMI.Config.PT.DBNC.AHHH;
   #HHHA.Config.HPT := #HMI.Config.PT.HLD.AHHH;
   #HHHA(IV := #Admin.SCL.SAIV,   // "HLR"
         HL := #HMI.Config.SP.Limits.HHH,
         H := #HMI.Config.SP.HYS.HHH,
         LR => #HMI.Alarm.AHHH);
END_REGION

REGION Network 58: High High Alarm
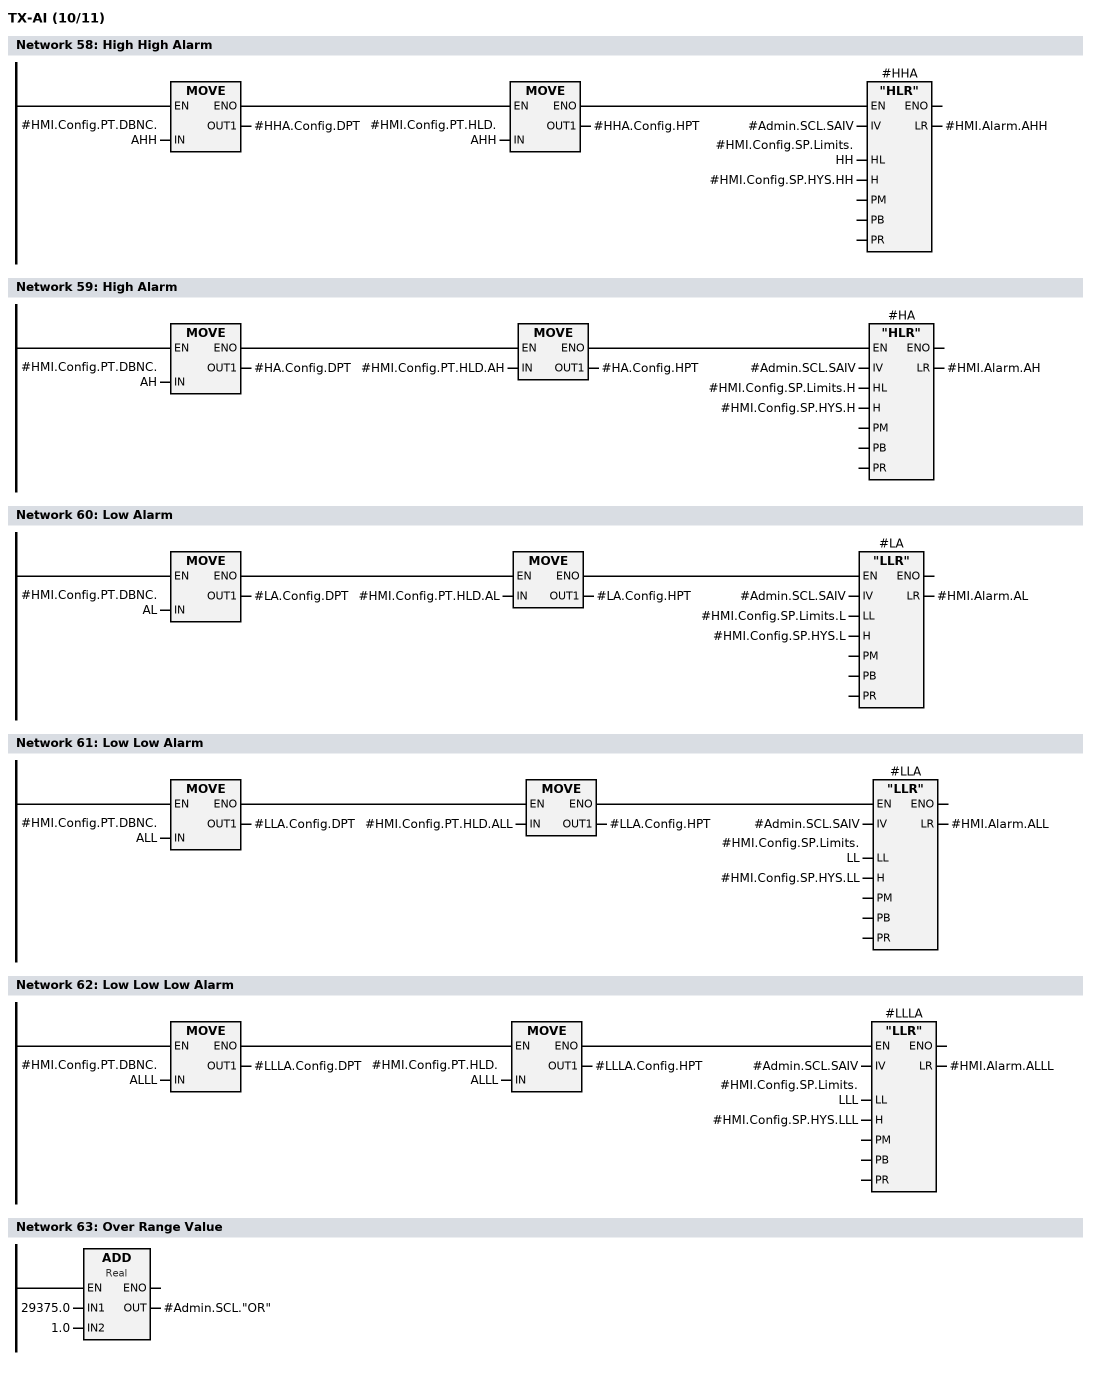
   RUNG wire#powerrail
      { S7_GenerateENO := "TRUE" } Move(in := #HMI.Config.PT.DBNC.AHH, out1 => #HHA.Config.DPT)
      { S7_GenerateENO := "TRUE" } Move(in := #HMI.Config.PT.HLD.AHH, out1 => #HHA.Config.HPT)
      #HHA(IV := #Admin.SCL.SAIV, HL := #HMI.Config.SP.Limits.HH, H := #HMI.Config.SP.HYS.HH, PM :=, PB :=, PR :=, LR => #HMI.Alarm.AHH)
   END_RUNG
   // the same network as SCL:
   // ENO of a box is taken as its EN; it also drops when the box reports an error
   #HHA.Config.DPT := #HMI.Config.PT.DBNC.AHH;
   #HHA.Config.HPT := #HMI.Config.PT.HLD.AHH;
   #HHA(IV := #Admin.SCL.SAIV, HL := #HMI.Config.SP.Limits.HH, H := #HMI.Config.SP.HYS.HH, LR => #HMI.Alarm.AHH);   // "HLR"
END_REGION

REGION Network 59: High Alarm
   RUNG wire#powerrail
      { S7_GenerateENO := "TRUE" } Move(in := #HMI.Config.PT.DBNC.AH, out1 => #HA.Config.DPT)
      { S7_GenerateENO := "TRUE" } Move(in := #HMI.Config.PT.HLD.AH, out1 => #HA.Config.HPT)
      #HA(IV := #Admin.SCL.SAIV, HL := #HMI.Config.SP.Limits.H, H := #HMI.Config.SP.HYS.H, PM :=, PB :=, PR :=, LR => #HMI.Alarm.AH)
   END_RUNG
   // the same network as SCL:
   // ENO of a box is taken as its EN; it also drops when the box reports an error
   #HA.Config.DPT := #HMI.Config.PT.DBNC.AH;
   #HA.Config.HPT := #HMI.Config.PT.HLD.AH;
   #HA(IV := #Admin.SCL.SAIV, HL := #HMI.Config.SP.Limits.H, H := #HMI.Config.SP.HYS.H, LR => #HMI.Alarm.AH);   // "HLR"
END_REGION

REGION Network 60: Low Alarm
   RUNG wire#powerrail
      { S7_GenerateENO := "TRUE" } Move(in := #HMI.Config.PT.DBNC.AL, out1 => #LA.Config.DPT)
      { S7_GenerateENO := "TRUE" } Move(in := #HMI.Config.PT.HLD.AL, out1 => #LA.Config.HPT)
      #LA(IV := #Admin.SCL.SAIV, LL := #HMI.Config.SP.Limits.L, H := #HMI.Config.SP.HYS.L, PM :=, PB :=, PR :=, LR => #HMI.Alarm.AL)
   END_RUNG
   // the same network as SCL:
   // ENO of a box is taken as its EN; it also drops when the box reports an error
   #LA.Config.DPT := #HMI.Config.PT.DBNC.AL;
   #LA.Config.HPT := #HMI.Config.PT.HLD.AL;
   #LA(IV := #Admin.SCL.SAIV, LL := #HMI.Config.SP.Limits.L, H := #HMI.Config.SP.HYS.L, LR => #HMI.Alarm.AL);   // "LLR"
END_REGION

REGION Network 61: Low Low Alarm
   RUNG wire#powerrail
      { S7_GenerateENO := "TRUE" } Move(in := #HMI.Config.PT.DBNC.ALL, out1 => #LLA.Config.DPT)
      { S7_GenerateENO := "TRUE" } Move(in := #HMI.Config.PT.HLD.ALL, out1 => #LLA.Config.HPT)
      #LLA(IV := #Admin.SCL.SAIV, LL := #HMI.Config.SP.Limits.LL, H := #HMI.Config.SP.HYS.LL, PM :=, PB :=, PR :=, LR => #HMI.Alarm.ALL)
   END_RUNG
   // the same network as SCL:
   // ENO of a box is taken as its EN; it also drops when the box reports an error
   #LLA.Config.DPT := #HMI.Config.PT.DBNC.ALL;
   #LLA.Config.HPT := #HMI.Config.PT.HLD.ALL;
   #LLA(IV := #Admin.SCL.SAIV, LL := #HMI.Config.SP.Limits.LL, H := #HMI.Config.SP.HYS.LL, LR => #HMI.Alarm.ALL);   // "LLR"
END_REGION

REGION Network 62: Low Low Low Alarm
   RUNG wire#powerrail
      { S7_GenerateENO := "TRUE" } Move(in := #HMI.Config.PT.DBNC.ALLL, out1 => #LLLA.Config.DPT)
      { S7_GenerateENO := "TRUE" } Move(in := #HMI.Config.PT.HLD.ALLL, out1 => #LLLA.Config.HPT)
      #LLLA(IV := #Admin.SCL.SAIV, LL := #HMI.Config.SP.Limits.LLL, H := #HMI.Config.SP.HYS.LLL, PM :=, PB :=, PR :=, LR => #HMI.Alarm.ALLL)
   END_RUNG
   // the same network as SCL:
   // ENO of a box is taken as its EN; it also drops when the box reports an error
   #LLLA.Config.DPT := #HMI.Config.PT.DBNC.ALLL;
   #LLLA.Config.HPT := #HMI.Config.PT.HLD.ALLL;
   #LLLA(IV := #Admin.SCL.SAIV,   // "LLR"
         LL := #HMI.Config.SP.Limits.LLL,
         H := #HMI.Config.SP.HYS.LLL,
         LR => #HMI.Alarm.ALLL);
END_REGION

REGION Network 63: Over Range Value
   RUNG wire#powerrail
      { S7_Templates := "SrcType := Real"; S7_GenerateENO := "TRUE" } Add(in1 := 29375.0, in2 := 1.0, out => #Admin.SCL."OR")
   END_RUNG
   // the same network as SCL:
   #Admin.SCL."OR" := 29375.0 + 1.0;
END_REGION

REGION Network 64: Under Range Value
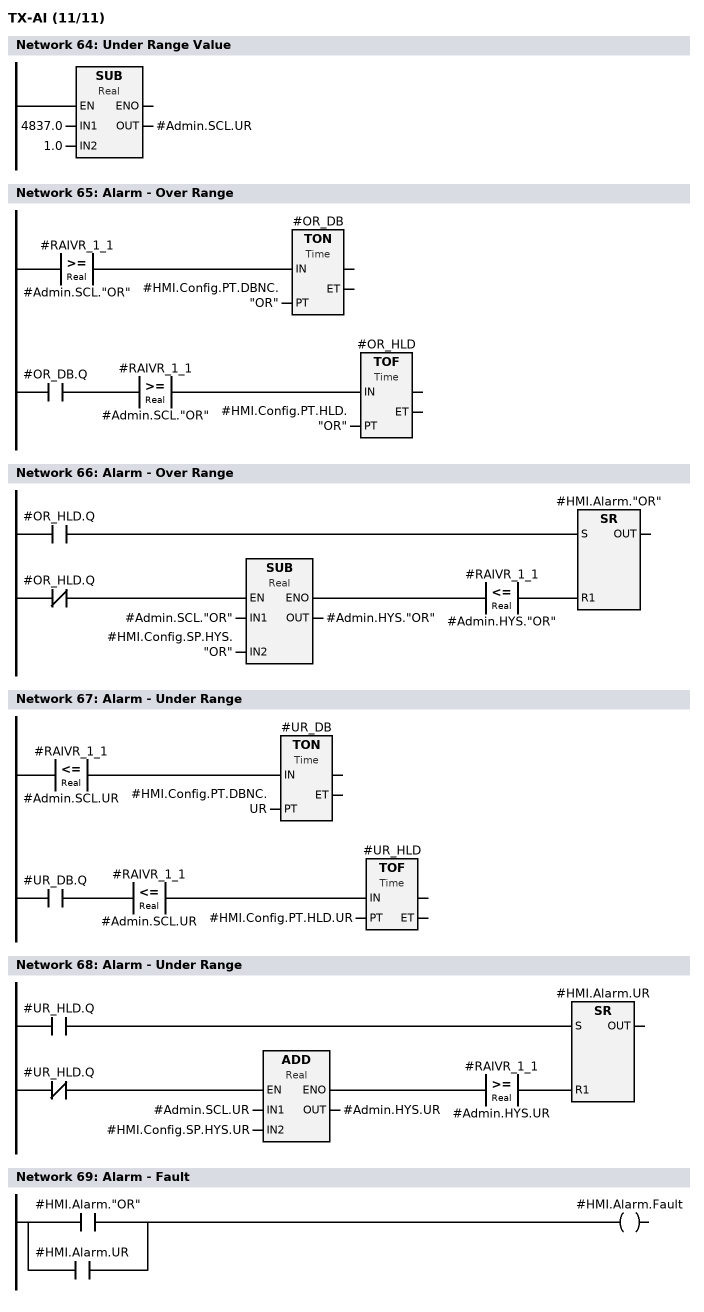
   RUNG wire#powerrail
      { S7_Templates := "SrcType := Real"; S7_GenerateENO := "TRUE" } Sub(in1 := 4837.0, in2 := 1.0, out => #Admin.SCL.UR)
   END_RUNG
   // the same network as SCL:
   #Admin.SCL.UR := 4837.0 - 1.0;
END_REGION

REGION Network 65: Alarm - Over Range
   RUNG wire#powerrail
      { S7_Templates := "SrcType := Real" } GE_Contact(in1 := #RAIVR_1_1, in2 := #Admin.SCL."OR")
      { S7_Templates := "time_type := Time" } #OR_DB.TON(pt := #HMI.Config.PT.DBNC."OR", et =>)
   END_RUNG
   RUNG wire#powerrail
      Contact( #OR_DB.Q )
      { S7_Templates := "SrcType := Real" } GE_Contact(in1 := #RAIVR_1_1, in2 := #Admin.SCL."OR")
      { S7_Templates := "time_type := Time" } #OR_HLD.TOF(pt := #HMI.Config.PT.HLD."OR", et =>)
   END_RUNG
   // the same network as SCL:
   #OR_DB(IN := #RAIVR_1_1 >= #Admin.SCL."OR", PT := #HMI.Config.PT.DBNC."OR");   // TON
   #OR_HLD(IN := #OR_DB.Q AND (#RAIVR_1_1 >= #Admin.SCL."OR"), PT := #HMI.Config.PT.HLD."OR");   // TOF
END_REGION

REGION Network 66: Alarm - Over Range
   RUNG wire#powerrail
      Contact( #OR_HLD.Q )
      S_SR(operand := #HMI.Alarm."OR", r1 := wire#w1)
   END_RUNG
   RUNG wire#powerrail
      I_Contact( #OR_HLD.Q )
      { S7_Templates := "SrcType := Real"; S7_GenerateENO := "TRUE" } Sub(in1 := #Admin.SCL."OR", in2 := #HMI.Config.SP.HYS."OR", out => #Admin.HYS."OR")
      { S7_Templates := "SrcType := Real" } LE_Contact(in1 := #RAIVR_1_1, in2 := #Admin.HYS."OR")
   END_RUNG wire#w1
   // the same network as SCL:
   // ENO of a box is taken as its EN; it also drops when the box reports an error
   IF NOT #OR_HLD.Q THEN #Admin.HYS."OR" := #Admin.SCL."OR" - #HMI.Config.SP.HYS."OR"; END_IF;
   IF #OR_HLD.Q THEN
       #HMI.Alarm."OR" := TRUE;   // SR flip-flop
   END_IF;
   IF NOT #OR_HLD.Q AND (#RAIVR_1_1 <= #Admin.HYS."OR") THEN #HMI.Alarm."OR" := FALSE; END_IF;
END_REGION

REGION Network 67: Alarm - Under Range
   RUNG wire#powerrail
      { S7_Templates := "SrcType := Real" } LE_Contact(in1 := #RAIVR_1_1, in2 := #Admin.SCL.UR)
      { S7_Templates := "time_type := Time" } #UR_DB.TON(pt := #HMI.Config.PT.DBNC.UR, et =>)
   END_RUNG
   RUNG wire#powerrail
      Contact( #UR_DB.Q )
      { S7_Templates := "SrcType := Real" } LE_Contact(in1 := #RAIVR_1_1, in2 := #Admin.SCL.UR)
      { S7_Templates := "time_type := Time" } #UR_HLD.TOF(pt := #HMI.Config.PT.HLD.UR, et =>)
   END_RUNG
   // the same network as SCL:
   #UR_DB(IN := #RAIVR_1_1 <= #Admin.SCL.UR, PT := #HMI.Config.PT.DBNC.UR);   // TON
   #UR_HLD(IN := #UR_DB.Q AND (#RAIVR_1_1 <= #Admin.SCL.UR), PT := #HMI.Config.PT.HLD.UR);   // TOF
END_REGION

REGION Network 68: Alarm - Under Range
   RUNG wire#powerrail
      Contact( #UR_HLD.Q )
      S_SR(operand := #HMI.Alarm.UR, r1 := wire#w1)
   END_RUNG
   RUNG wire#powerrail
      I_Contact( #UR_HLD.Q )
      { S7_Templates := "SrcType := Real"; S7_GenerateENO := "TRUE" } Add(in1 := #Admin.SCL.UR, in2 := #HMI.Config.SP.HYS.UR, out => #Admin.HYS.UR)
      { S7_Templates := "SrcType := Real" } GE_Contact(in1 := #RAIVR_1_1, in2 := #Admin.HYS.UR)
   END_RUNG wire#w1
   // the same network as SCL:
   // ENO of a box is taken as its EN; it also drops when the box reports an error
   IF NOT #UR_HLD.Q THEN #Admin.HYS.UR := #Admin.SCL.UR + #HMI.Config.SP.HYS.UR; END_IF;
   IF #UR_HLD.Q THEN
       #HMI.Alarm.UR := TRUE;   // SR flip-flop
   END_IF;
   IF NOT #UR_HLD.Q AND (#RAIVR_1_1 >= #Admin.HYS.UR) THEN #HMI.Alarm.UR := FALSE; END_IF;
END_REGION

REGION Network 69: Alarm - Fault
   RUNG wire#powerrail
      Contact( #HMI.Alarm."OR" )
      wire#w1
      Coil( #HMI.Alarm.Fault )
   END_RUNG
   RUNG wire#powerrail
      Contact( #HMI.Alarm.UR )
   END_RUNG wire#w1
   // the same network as SCL:
   #HMI.Alarm.Fault := #HMI.Alarm."OR" OR #HMI.Alarm.UR;
END_REGION
END_FUNCTION_BLOCK
